{attribute addProperty BoxType "EPP1321-0060-0016"}
{attribute addProperty Id "A_0019_EPP1322_0001_0016A_0019_EPP1322_0001_0016_DC7CEC292816352"}
{attribute addProperty CRC "3773210807"}
{attribute addProperty SizeInBites "2816"}
{attribute addProperty SizeInBytes "352"}
TYPE A_0018_EPP1321_0060_0016_E0E6A0B7 EXTENDS EPP1321_179A0949 :
STRUCT
	{attribute addProperty Name "A_0019_EPP1322_0001_0016"}
	A_0019_EPP1322_0001_0016 : A_0019_EPP1322_0001_0016_DC7CEC29;
END_STRUCT
END_TYPE

(* stored: Version 1.2.0.0, ProductVersion 3.1.4024.9
   DUT A_0018_EPP1321_0060_0016_E0E6A0B7: Id {c16eddac-2c2f-4b6f-b499-0a96a1418f22} *)
